// SIMATIC S7-200 project (STEP 7-Micro/WIN), CPU 224 REL 01.11

SYMBOL_TABLE USER1
NUT_NHAN         I0.0
CD1              Q1.0
CD2              Q1.1
X1               Q0.0
V1               Q0.1
D1               Q0.2
X2               Q0.3
V2               Q0.4
D2               Q0.5
MODE             M0.0
DUY_TRI          M0.1
END_SYMBOL_TABLE

ORGANIZATION_BLOCK MAIN:OB1
TITLE=PROGRAM COMMENTS
BEGIN
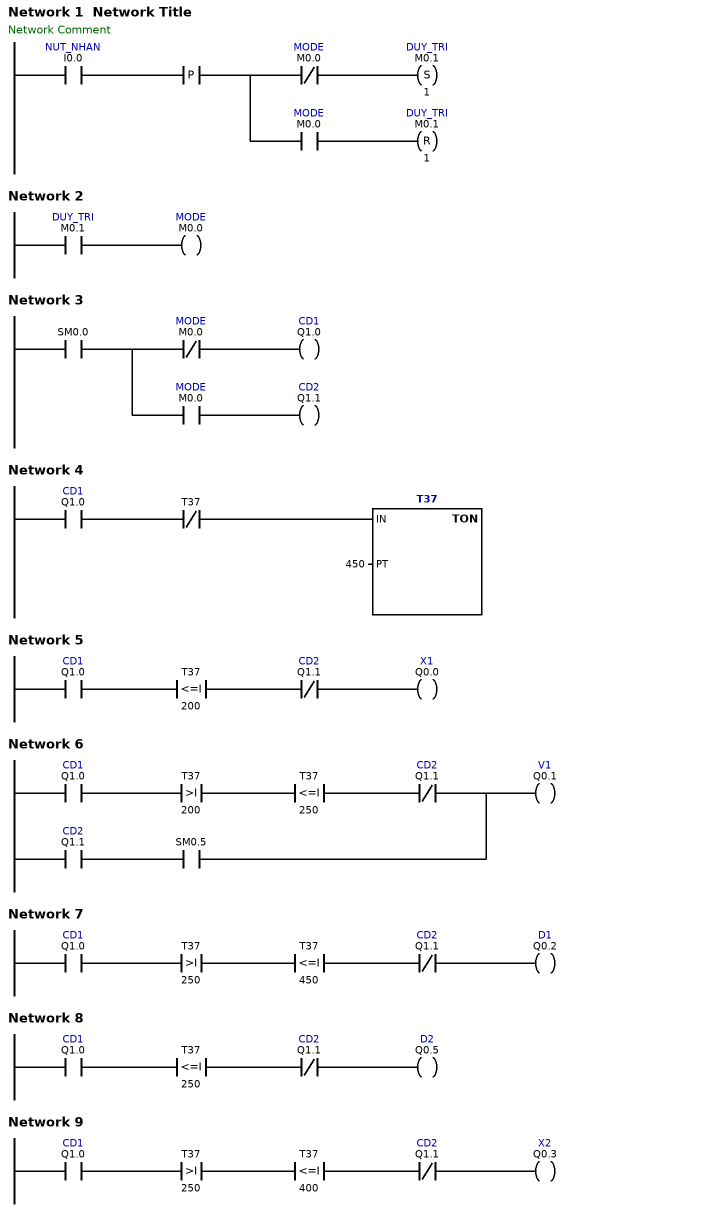
Network 1 // Network Title
// Network Comment
LD     NUT_NHAN:I0.0
EU
LPS
AN     MODE:M0.0
S      DUY_TRI:M0.1, 1
LPP
A      MODE:M0.0
R      DUY_TRI:M0.1, 1
Network 2
LD     DUY_TRI:M0.1
=      MODE:M0.0
Network 3
LD     SM0.0
LPS
AN     MODE:M0.0
=      CD1:Q1.0
LPP
A      MODE:M0.0
=      CD2:Q1.1
Network 4
LD     CD1:Q1.0
AN     T37
TON    T37, 450
Network 5
LD     CD1:Q1.0
AW<=   T37, 200
AN     CD2:Q1.1
=      X1:Q0.0
Network 6
LD     CD1:Q1.0
AW>    T37, 200
AW<=   T37, 250
AN     CD2:Q1.1
LD     CD2:Q1.1
A      SM0.5
OLD
=      V1:Q0.1
Network 7
LD     CD1:Q1.0
AW>    T37, 250
AW<=   T37, 450
AN     CD2:Q1.1
=      D1:Q0.2
Network 8
LD     CD1:Q1.0
AW<=   T37, 250
AN     CD2:Q1.1
=      D2:Q0.5
Network 9
LD     CD1:Q1.0
AW>    T37, 250
AW<=   T37, 400
AN     CD2:Q1.1
=      X2:Q0.3
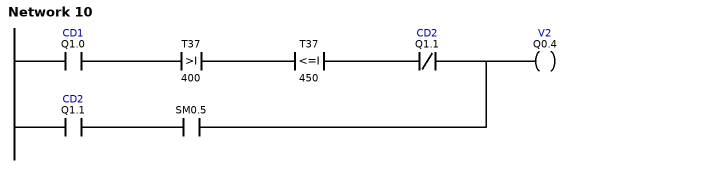
Network 10
LD     CD1:Q1.0
AW>    T37, 400
AW<=   T37, 450
AN     CD2:Q1.1
LD     CD2:Q1.1
A      SM0.5
OLD
=      V2:Q0.4
END_ORGANIZATION_BLOCK
